FUNCTION_BLOCK FB_LeakTester IMPLEMENTS I_LeakTester
VAR_INPUT
END_VAR
VAR_OUTPUT
END_VAR
VAR
END_VAR

{warning 'add method implementation '}
METHOD ParamRead
END_METHOD

{warning 'add method implementation '}
METHOD ParamWrite
END_METHOD

{warning 'add method implementation '}
METHOD PollResult : BOOL
END_METHOD

{warning 'add method implementation '}
METHOD ProgramSelect : INT
END_METHOD

{warning 'add method implementation '}
METHOD ProgramStart : BOOL
END_METHOD

{warning 'add method implementation '}
METHOD ProgramStop : BOOL
END_METHOD

{warning 'add method implementation '}
METHOD Zero : BOOL
END_METHOD

END_FUNCTION_BLOCK

(* stored: Version 1.1.0.1, ProductVersion 3.1.4024.15
   POU FB_LeakTester: Id {8d80e9d5-1c82-40d0-9db4-b193c6d348d1}, SpecialFunc None
   Method ParamRead: Id {4883de8a-6c73-42a0-a2e1-ec4689d0afc5}
   Method ParamWrite: Id {b5d71b41-70dc-484c-b001-2324bc8bf155}
   Method PollResult: Id {93b9b3ea-8a1b-49a8-a1e2-581217cffea1}
   Method ProgramSelect: Id {2bfc00f6-6b89-47be-afac-8f9673ddd020}
   Method ProgramStart: Id {0ba957ed-38a8-4e73-8123-eb3af5b8d31e}
   Method ProgramStop: Id {55be82be-20a5-45e6-8f17-50be61f6dd34}
   Method Zero: Id {fdea39eb-dbff-442c-a634-1b374c255bbd} *)
